// TIA Portal V20 export
TYPE "PII - VDM28-50-R1-IO"
   STRUCT
      "Process Data Input - Distance (16 bit)" : Word;
   END_STRUCT;
END_TYPE
